// TIA Portal V19 export
TYPE "TrkMng_Row"
   STRUCT
      Visible : Bool;
      RowColor : Int;
      PNum : Int;
      IDPiece : UDInt;
      PartProgram : DInt;
      Sum_Result : "Trk_AreaResult";
   END_STRUCT;
END_TYPE
